RoboDK station: UR robot with rail.rdk

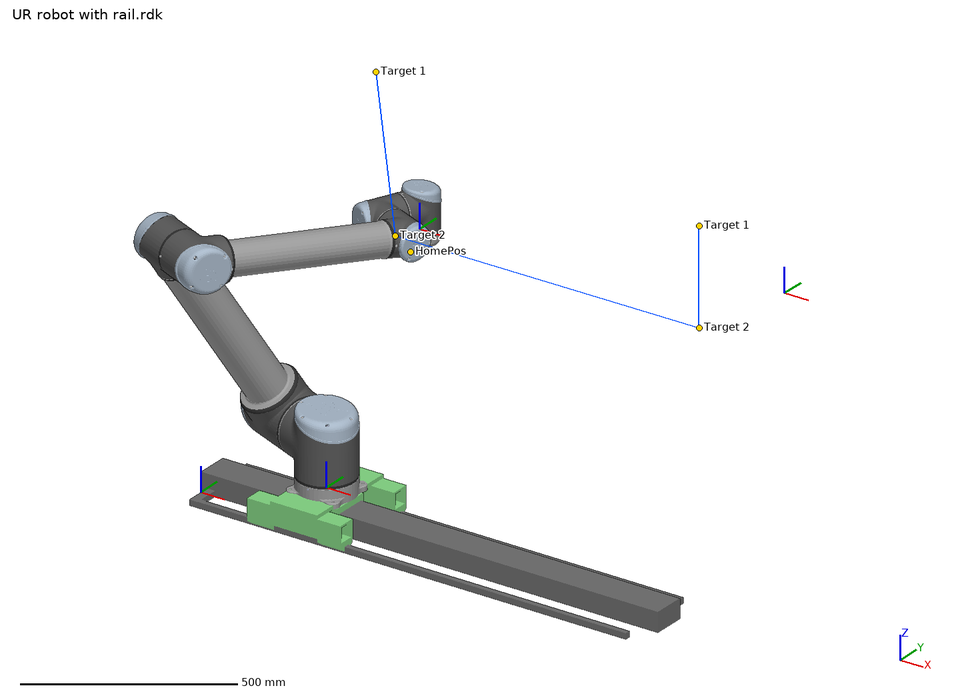
[picture v0: the station drawn from its stored meshes, robots at their saved joint values, targets as dots, program paths as lines]
Station test. Poses are relative to the parent item; angles as X-Y-Z fixed-axis rotations.
  - frame FL linear rail-930 Base at (-911.43, 0, 0) mm
    - robot FL linear rail-930: 1 axes
        modified DH rows (alpha deg, a mm, theta deg, d mm): 0, 0, 0, 0 linear
        base shift (0, 0, 0) mm, rotated rx 0 ry 90 rz 0 deg
        joint limits [0] to [930]; home [0]; saved at [151.19]
      - frame UR10 Base at (0, 0, 0) mm
        - robot UR10: 6 axes, payload 10 kg, reach 1300 mm, repeatability 0.1 mm, weight 28.9 kg
            modified DH rows (alpha deg, a mm, theta deg, d mm): 0, 0, 0, 118; 90, 0, 180, 0; 0, 612.7, 0, 0; 0, 571.6, 0, 163.9; -90, 0, 0, 115.7; 90, 0, 180, 92.2
            joint limits [-360, -360, -360, -360, -360, -360] to [360, 360, 360, 360, 360, 360]; home [0, -90, 90, 0, 90, 0]; saved at [-113.208, -122.043, 129.907, -97.42, -90.19, 156.793]
        - target HomePos (joint target) at (-10.02, 351.8, 458.46) mm, rotated rx 90 ry 0 rz -180 deg; joints [-126.907, -127.042, 130.341, -3.299, 53.093, 0] of UR10
    - target RailPos1 (joint target) at (170.4, 44, 84) mm; joints [0] of FL linear rail-930
    - target RailPos2 (joint target) at (1100.4, 44, 84) mm; joints [930, 0, 0, 0, 0, 0] of FL linear rail-930
    - frame Reference 1 at (0, 875.24, 322.36) mm
      - target Target 1 (Cartesian target) at (6.5, -184.49, 475.77) mm, rotated rx 170.25 ry 0.38 rz -177.79 deg; joints [-33.196, -178.793, 130.778, -47.365, -98.155, 234.182] of UR10
      - target Target 2 (Cartesian target) at (6.5, -107.2, 26.42) mm, rotated rx 170.25 ry 0.38 rz -177.79 deg; joints [-90, -74.736, 115.477, -140.5, -90, 177.762] of UR10
    - frame Reference 2 at (1373.34, 373.2, 743.21) mm
      - target Target 1 (Cartesian target) at (-282.95, 62.59, 66.84) mm, rotated rx -179.52 ry 0 rz -180 deg; joints [-47.042, -84.407, 168.001, -173.24, -89.671, 222.957] of UR10
      - target Target 2 (Cartesian target) at (-282.95, 62.59, -193.16) mm, rotated rx -179.52 ry 0 rz -180 deg; joints [-47.042, -8.216, 155.872, -237.302, -89.671, 222.957] of UR10
  - program MoveRailPos1 (1 instructions, listed below)
  - program MoveRailPos2 (1 instructions, listed below)
  - program GoHomePos (2 instructions, listed below)
  - program MainProgram (9 instructions, listed below)
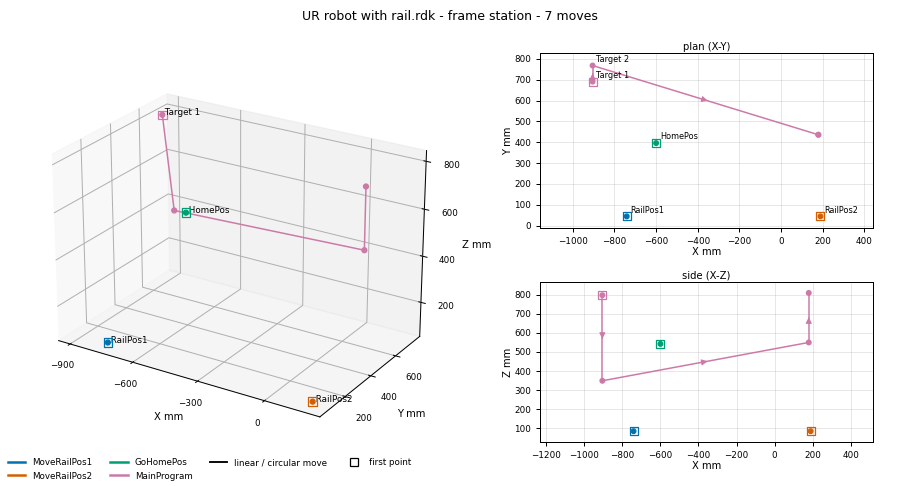
[picture p0: tool path of UR robot with rail.rdk in frame station, 7 of 7 moves have a stored position in this frame; points joined in program order, loops and branches not executed]

--- program MoveRailPos1 (robot FL linear rail-930) ---
  MoveJ (RailPos1)

--- program MoveRailPos2 (robot FL linear rail-930) ---
  MoveJ (RailPos2)

--- program GoHomePos (robot UR10) ---
  Set Ref.: UR10 Base
  MoveJ (HomePos)

--- program MainProgram (robot UR10) ---
  Call GoHomePos
  Call MoveRailPos1
  Set Ref.: Reference 1
  MoveJ (Target 1)
  MoveL (Target 2)
  Call MoveRailPos2
  Set Ref.: Reference 2
  MoveL (Target 2)
  MoveL (Target 1)
